TYPE ST_System_BSp_Verb_Stellwert :
STRUCT
	Anford_Pumpe	: BOOL;

	Einschaltperiode_Max	: TIME := T#10S;
	Einschalten				: BOOL;
END_STRUCT
END_TYPE

(* stored: Version 1.1.0.1, ProductVersion 3.1.4024.9
   DUT ST_System_BSp_Verb_Stellwert: Id {a96044c0-f391-44e9-9f42-7effc1cb9ab5} *)
